// TIA Portal V19 export
TYPE "LAF_typeEmControlNode"
// Control node of the equipment module
// stored: Access Published
   STRUCT
      commands : "LAF_typeEmCommands";
      status { ExternalWritable := 'False'} : "LAF_typeEmStatus";
   END_STRUCT;
END_TYPE
